Fanuc KAREL source: kt00110.KL

-- PROVISIONAL review KL for V1013-1; original PC SHA256 9039b2363a12013e963ddf26c7678e2b382831f7048501c63e32143decb19346
-- Incomplete behavior may be omitted. Consult companion uncertainty JSON. Do not deploy.
PROGRAM KT00110
%NOLOCKGROUP
VAR
  R1 : REAL
  OUT : REAL
-- UNRESOLVED_DECL Y2 type=002018
BEGIN
  -- UNRESOLVED_PC offsets 5-16; opcodes 2E,23
  -- UNRESOLVED_PC offsets 21-35; opcodes 2E,22,9D,33,B2
  -- UNRESOLVED_PC offsets 40-63; opcodes 21,22,9D,33,B1,64,6C,23
  -- UNRESOLVED_PC offsets 68-72; opcodes 7F
END KT00110
